(* IEC 61131-3 sources: RL_MAR/experiments/comparison/llm4plc/results/gpt-4o-mini_20260506_100619/20260506_101158, 4 files *)

(* ---- generated_code_iteration_0.st ---- *)
ructured-text
FUNCTION_BLOCK FB_MergeBytes
VAR_INPUT
    byteArray : ARRAY[1..20] OF DINT; (* Byte array to be merged *)
END_VAR
VAR_OUTPUT
    dwordArray : ARRAY[1..10] OF DINT; (* Merged double word array *)
    mergeDwordNum : DINT; (* Actual number of merged double words *)
END_VAR
VAR
    i, j, k : INT; (* Index variables *)
    tempDword : DINT; (* Temporary variable to hold merged double word *)
END_VAR
VAR CONSTANT
    BYTE_ARRAY_SIZE : DINT := 20; (* Size of the input byte array *)
    DWORD_ARRAY_SIZE : DINT := 10; (* Size of the output DINT array *)
END_VAR

(* Initialize state variables *)
i := 1;
j := 1;
k := 0;
mergeDwordNum := 0;

(* Initialize dwordArray to zero *)
FOR j := 1 TO DWORD_ARRAY_SIZE DO
    dwordArray[j] := 0;
END_FOR

(* Merging bytes into double words *)
WHILE (i <= BYTE_ARRAY_SIZE) AND (j <= DWORD_ARRAY_SIZE) DO
    IF (i + 3 <= BYTE_ARRAY_SIZE) THEN
        tempDword := byteArray[i] + (byteArray[i + 1] << 8) + (byteArray[i + 2] << 16) + (byteArray[i + 3] << 24);
        dwordArray[j] := tempDword;
        mergeDwordNum := mergeDwordNum + 1;
        j := j + 1;
        i := i + 4;
    ELSE
        EXIT; (* Exit loop if not enough bytes left to merge *)
    END_IF
END_WHILE

END_FUNCTION_BLOCK

(* ---- generated_code_iteration_1.st ---- *)
START_REASON
The errors in the original Structured Text (ST) code primarily stem from the use of the bitwise left shift operator (`<<`) which is not supported in the CODESYS environment for the merging of bytes into double words. Instead, expressions should be used to achieve the same result without the bitwise operations. Additionally, the variable sections should be properly closed with `END_VAR` instead of `END_VAR_OUTPUT` or `END_VAR_INPUT`.
END_REASON

START_ST
FUNCTION_BLOCK FB_MergeBytes
VAR_INPUT
    byteArray : ARRAY[1..20] OF DINT; (* Byte array to be merged *)
END_VAR
VAR_OUTPUT
    dwordArray : ARRAY[1..10] OF DINT; (* Merged double word array *)
    mergeDwordNum : DINT; (* Actual number of merged double words *)
END_VAR
VAR
    i, j : INT; (* Index variables *)
    tempDword : DINT; (* Temporary variable to hold merged double word *)
END_VAR
VAR CONSTANT
    BYTE_ARRAY_SIZE : DINT := 20; (* Size of the input byte array *)
    DWORD_ARRAY_SIZE : DINT := 10; (* Size of the output DINT array *)
END_VAR

(* Initialize state variables *)
i := 1;
j := 1;
mergeDwordNum := 0;

(* Initialize dwordArray to zero *)
FOR j := 1 TO DWORD_ARRAY_SIZE DO
    dwordArray[j] := 0;
END_FOR

(* Merging bytes into double words *)
WHILE (i <= BYTE_ARRAY_SIZE) AND (j <= DWORD_ARRAY_SIZE) DO
    IF (i + 3 <= BYTE_ARRAY_SIZE) THEN
        tempDword := byteArray[i] + (byteArray[i + 1] * 256) + (byteArray[i + 2] * 65536) + (byteArray[i + 3] * 16777216);
        dwordArray[j] := tempDword;
        mergeDwordNum := mergeDwordNum + 1;
        j := j + 1;
        i := i + 4;
    ELSE
        EXIT; (* Exit loop if not enough bytes left to merge *)
    END_IF
END_WHILE

END_FUNCTION_BLOCK
END_ST

(* ---- generated_code_iteration_2.st ---- *)
START_REASON
The errors in the original Structured Text (ST) code were primarily caused by the use of the wrong data type for the `byteArray` variable. The `byteArray` was defined as an array of `DINT`, which is not suitable for holding byte values. Instead, it should be defined as an array of `BYTE`. Additionally, the merging logic needs to ensure that the correct data types are used throughout the calculations. The output variable `dwordArray` should remain as `DINT` since it is meant to hold merged double words. The variable sections should be properly closed with `END_VAR` instead of `END_VAR_OUTPUT` or `END_VAR_INPUT`.
END_REASON

START_ST
FUNCTION_BLOCK FB_MergeBytes
VAR_INPUT
    byteArray : ARRAY[1..20] OF BYTE; (* Byte array to be merged *)
END_VAR
VAR_OUTPUT
    dwordArray : ARRAY[1..10] OF DINT; (* Merged double word array *)
    mergeDwordNum : DINT; (* Actual number of merged double words *)
END_VAR
VAR
    i, j : INT; (* Index variables *)
    tempDword : DINT; (* Temporary variable to hold merged double word *)
END_VAR
VAR CONSTANT
    BYTE_ARRAY_SIZE : DINT := 20; (* Size of the input byte array *)
    DWORD_ARRAY_SIZE : DINT := 10; (* Size of the output DINT array *)
END_VAR

(* Initialize state variables *)
i := 1;
j := 1;
mergeDwordNum := 0;

(* Initialize dwordArray to zero *)
FOR j := 1 TO DWORD_ARRAY_SIZE DO
    dwordArray[j] := 0;
END_FOR

(* Merging bytes into double words *)
WHILE (i <= BYTE_ARRAY_SIZE) AND (j <= DWORD_ARRAY_SIZE) DO
    IF (i + 3 <= BYTE_ARRAY_SIZE) THEN
        tempDword := DINT(byteArray[i]) + (DINT(byteArray[i + 1]) * 256) + (DINT(byteArray[i + 2]) * 65536) + (DINT(byteArray[i + 3]) * 16777216);
        dwordArray[j] := tempDword;
        mergeDwordNum := mergeDwordNum + 1;
        j := j + 1;
        i := i + 4;
    ELSE
        EXIT; (* Exit loop if not enough bytes left to merge *)
    END_IF
END_WHILE

END_FUNCTION_BLOCK
END_ST

(* ---- generated_code_iteration_3.st ---- *)
START_REASON
The errors in the original Structured Text (ST) code were primarily due to the incorrect use of the `DINT` keyword in the variable declarations and assignments. Specifically, the feedback indicated that the `DINT` keyword should be replaced with a semicolon (`;`) to properly terminate statements. This suggests that there were syntax issues in the code that needed to be corrected. Additionally, the variable sections should be properly closed with `END_VAR` instead of `END_VAR_OUTPUT` or `END_VAR_INPUT`. I will ensure that the code adheres to these requirements and correct any syntax errors.
END_REASON

START_ST
FUNCTION_BLOCK FB_MergeBytes
VAR_INPUT
    byteArray : ARRAY[1..20] OF BYTE; (* Byte array to be merged *)
END_VAR
VAR_OUTPUT
    dwordArray : ARRAY[1..10] OF DINT; (* Merged double word array *)
    mergeDwordNum : DINT; (* Actual number of merged double words *)
END_VAR
VAR
    i, j : INT; (* Index variables *)
    tempDword : DINT; (* Temporary variable to hold merged double word *)
END_VAR
VAR CONSTANT
    BYTE_ARRAY_SIZE : DINT := 20; (* Size of the input byte array *)
    DWORD_ARRAY_SIZE : DINT := 10; (* Size of the output DINT array *)
END_VAR

(* Initialize state variables *)
i := 1;
j := 1;
mergeDwordNum := 0;

(* Initialize dwordArray to zero *)
FOR j := 1 TO DWORD_ARRAY_SIZE DO
    dwordArray[j] := 0;
END_FOR

(* Merging bytes into double words *)
WHILE (i <= BYTE_ARRAY_SIZE) AND (j <= DWORD_ARRAY_SIZE) DO
    IF (i + 3 <= BYTE_ARRAY_SIZE) THEN
        tempDword := BYTE_TO_DINT(byteArray[i]) + (BYTE_TO_DINT(byteArray[i + 1]) * 256) + (BYTE_TO_DINT(byteArray[i + 2]) * 65536) + (BYTE_TO_DINT(byteArray[i + 3]) * 16777216);
        dwordArray[j] := tempDword;
        mergeDwordNum := mergeDwordNum + 1;
        j := j + 1;
        i := i + 4;
    ELSE
        EXIT; (* Exit loop if not enough bytes left to merge *)
    END_IF
END_WHILE

END_FUNCTION_BLOCK
END_ST
